{attribute 'linkalways'} 
{attribute 'no_explicit_call' := 'This FB is a CLASS and must be accessed using methods or properties'}
{attribute 'enable_dynamic_creation'}
FUNCTION_BLOCK FINAL Node_DigitalOutput EXTENDS HardwareNode
VAR
	output AT %Q* : BOOL;
	in : _BOOL(FALSE);
END_VAR

METHOD FB_init : BOOL
VAR_INPUT
	bInitRetains : BOOL; // if TRUE, the retain variables are initialized (warm start / cold start)
	bInCopyCode : BOOL;  // if TRUE, the instance afterwards gets moved into the copy code (online change)
END_VAR
AddInput('in', in);
END_METHOD

METHOD PROTECTED OnExecute
VAR
END_VAR
output := in.Value;
END_METHOD

END_FUNCTION_BLOCK

(* stored: Version 1.1.0.1, ProductVersion 3.1.4024.13
   POU Node_DigitalOutput: Id {8eb2478b-dfad-4133-8e9b-5cd4ecfbbad8}, SpecialFunc None
   Folder Constructor: Id {181531a4-5453-4c8e-8722-585931b10bf9}
   Method FB_init: Id {c123118c-9d74-4bb9-9311-7cac55c8109b}
   Method OnExecute: Id {68571122-a377-4d1a-96e4-62df1bbbcbe5} *)
